{attribute 'qualified_only'}
{attribute 'strict'}
{attribute 'to_string'}
TYPE E_TowerLamp :
(
	OFF, //대기상태 (Signal)
	RED, // Alarm
	YELLOW, // Warning
	GREEN, // Running
	BLUE, // Maint
	WHITE, // Idle
	BUZZER
):= OFF;
END_TYPE

(* stored: Version 1.1.0.1, ProductVersion 3.1.4026.11
   DUT E_TowerLamp: Id {e86f6cd1-f9e6-45eb-a187-c4714b576caf} *)
